INTERFACE I_SeasonState EXTENDS I_State

PROPERTY bRaining : BOOL
GET
END_GET
END_PROPERTY

PROPERTY bSnowing : BOOL
GET
END_GET
END_PROPERTY

PROPERTY bSunShining : BOOL
GET
END_GET
END_PROPERTY

PROPERTY bWindBlowing : BOOL
GET
END_GET
END_PROPERTY

METHOD ChangeToSummerTyres
VAR_INPUT
END_VAR
END_METHOD

METHOD ChangeToWinterTyres
VAR_INPUT
END_VAR
END_METHOD

PROPERTY eState : E_Season
GET
END_GET
END_PROPERTY

METHOD ABSTRACT NextSeason
VAR_INPUT
END_VAR
END_METHOD

PROPERTY nLeavesState : BYTE
GET
END_GET
END_PROPERTY

PROPERTY nTyresType : BYTE
GET
END_GET
END_PROPERTY

PROPERTY sState : STRING(MAX_STRING_LENGTH)
GET
END_GET
END_PROPERTY

END_INTERFACE

(* stored: Version 1.1.0.1, ProductVersion 3.1.4024.12
   Itf I_SeasonState: Id {00b7b34e-1219-4d25-8b3f-b4a9937d836d}
   Folder Properties: Id {2c6ac8ec-4efc-4064-8a71-36a73796ff6a}
   Property bRaining: Id {cddc6117-6d17-475a-88b7-10bea0a71212}
   Get Get: Id {c30a5975-bb3d-460d-9642-c2e21e4fac09}
   Property bSnowing: Id {80bb9182-dc75-4675-ac9f-96823f5b35f2}
   Get Get: Id {6858f2d2-c318-4def-a47c-01769fd2c447}
   Property bSunShining: Id {b94c867a-9207-44b9-9bcd-f64d0bc805a7}
   Get Get: Id {a14cef2f-af4b-4c9a-b19c-9af71240ff6b}
   Property bWindBlowing: Id {454e404d-1a89-4b60-8998-94a44092832a}
   Get Get: Id {2739f058-c4ec-4d3a-a7ef-333019e28a9b}
   Method ChangeToSummerTyres: Id {f42224d7-7bb6-4f96-abd1-2ebff2ba037a}
   Method ChangeToWinterTyres: Id {ffcdac36-ceb5-49de-b985-aa96f23234d8}
   Property eState: Id {61772e44-0544-4fd3-ad55-472f34944e3a}
   Get Get: Id {61563538-ca5e-4561-927f-9a6e4393aab9}
   Method NextSeason: Id {f4f336ec-09b1-4cf4-bcfc-6498d0191315}
   Property nLeavesState: Id {3e980e0e-56df-4f55-8657-f97f6c149753}
   Get Get: Id {6859c9bc-ac40-478e-a3b8-a4b8132b8fb2}
   Property nTyresType: Id {539217fb-42dd-430f-a135-6cc10f0df4cf}
   Get Get: Id {e5a96458-e1ea-413c-adb3-ebe745781436}
   Property sState: Id {eb6713cb-bad6-4a0d-99c5-8e6abb7e08d9}
   Get Get: Id {cb7c060f-c6b8-4baa-995d-6c401e49b52c} *)
